TYPE CmpConvMergeConfig :
STRUCT
	BufferSensorOnTime: TIME;
	BufferSensorOffTime: TIME;
	MergeTimeSpacing: TIME;
	MergeTimeMainTravel: TIME;
	MergeTimeSpurTravel: TIME;
	UseReleaseRatio: BOOL;
	RatioMain: REAL;
	RatioSpur: REAL;
END_STRUCT
END_TYPE

(* stored: Version 1.1.0.1, ProductVersion 3.1.4024.6
   DUT CmpConvMergeConfig: Id {44f908bb-9040-4cd2-b08f-951fa0fa96af} *)
